(* CODESYS project Kurgan.project
   Company: Plinfa
   Title: Burner
   Author: Serhii Surmylo
   Version: 0.0.0.0

Project tree, tasks and I/O mapping:
  MyController : TM241CEC24T/U, Schneider Electric, order no. TM241CEC24T/U, version 4.0.5.9
    application Application
      task MAST (cyclic, interval 20 ms, priority 15, watchdog 100 ms x 1) calls POU_test
      global variables GVL
      program POU_test [LD]
      Symbols
      function block POU [LD]
    DI : Digital Inputs, Schneider Electric, version 4.0.5.9
        input  A1_IW0 : WORD  // IW0
        input  ibDI_IB1 : BYTE  // IB1
    DQ : Digital Outputs, Schneider Electric, version 4.0.5.9
        output A1_QW0 : WORD  // QW0
        output qbDQ_QB1 : BYTE  // QB1
    Counters : Counters, Schneider Electric, version 4.0.5.9
    Pulse_Generators : Pulse Generators, Schneider Electric, version 4.0.5.9
    Cartridge_1 : Cartridge, Schneider Electric, version 4.0.5.9
    IO_Bus : IO bus - TM3, Schneider Electric, version 4.0.5.9
      A3 : TM2AMI8HT, Schneider Electric, order no. TM2AMI8HT, version 3.1.2.14
          input  A3_IW0 : INT  // IW0
          input  A3_IW1 : INT  // IW1
          input  A3_IW2 : INT  // IW2
          input  A3_IW3 : INT  // IW3
          input  A3_IW4 : INT  // IW4
          input  A3_IW5 : INT  // IW5
          input  A3_IW6 : INT  // IW6
          input  A3_IW7 : INT  // IW7
      A4 : TM2AMI8HT, Schneider Electric, order no. TM2AMI8HT, version 3.1.2.14
          input  A4_IW0 : INT  // IW0
          input  A4_IW1 : INT  // IW1
          input  A4_IW2 : INT  // IW2
          input  A4_IW3 : INT  // IW3
          input  A4_IW4 : INT  // IW4
          input  A4_IW5 : INT  // IW5
          input  A4_IW6 : INT  // IW6
          input  A4_IW7 : INT  // IW7
      A2 : TM3DQ32TK, Schneider Electric, order no. TM3DQ32TK, version 1.0.1.2
          output A2_QD1 : DWORD  // QD0
      A5 : TM2ARI8LT, Schneider Electric, order no. TM2ARI8LT, version 3.1.1.14
          input  A5_IW0 : INT  // IW0
          input  A5_IW1 : INT  // IW1
          input  A5_IW2 : INT  // IW2
          input  A5_IW3 : INT  // IW3
          input  A5_IW4 : INT  // IW4
          input  A5_IW5 : INT  // IW5
          input  A5_IW6 : INT  // IW6
          input  A5_IW7 : INT  // IW7
    COM_Bus : COM bus, Schneider Electric, version 4.0.5.9
    Ethernet_1 : Ethernet Network, Schneider Electric, version 4.0.5.9
        settings: IPAddress = [192, 168, 0, 10]; SubnetMask = [255, 255, 255, 0]; GatewayAddress = [192, 168, 0, 1]; WebServer = TRUE; FTP Server = TRUE; SoMachine Protocol = TRUE; Modbus Server = TRUE; NetManage Protocol = TRUE; SNMP protocol = TRUE; Enable Routing = FALSE; WebVisu protocol = TRUE; DHCP Server Active = TRUE
    Serial_Line_1 : Serial line, Schneider Electric, version 4.0.5.9
    Serial_Line_2 : Serial line, Schneider Electric, version 4.0.5.9
    CAN_1 : CANopen bus, Schneider Electric, version 4.0.5.9
  HMIGTO5310_5315 : HMIGTO5310/5315, Schneider Electric, order no. HMIGTO5310/5315, version 3.5.3.55
    HMI Application
    COM1
      SoMachine_Network_Manager : SoMachine-Network Manager, Schneider Electric, version 4.0.0.2
    COM2
      SoMachine_Network_Manager1 : SoMachine-Network Manager, Schneider Electric, version 4.0.0.2
    Ethernet
      SoMachine_Network_Manager2 : SoMachine-Network Manager, Schneider Electric, version 4.0.0.2
    USB
      SoMachine_Network_Manager3 : SoMachine-Network Manager, Schneider Electric, version 4.0.0.2
  program POU_modbus_SINGLE_WRITE [LD]
  program POU_modbus_READ_VAR [LD]
  program POU_modbus_WRITE_VAR_bit [FBD]
  Vijeo Designer Project Container Data
  Vijeo Designer Project Container
*)

// MyController/Application/GVL
VAR_GLOBAL
END_VAR
VAR_GLOBAL
	KLxx_0_1: BOOL;
	KLxx_ON_OFF: BOOL;
END_VAR

// MyController/Application/POU_test
PROGRAM POU_test
VAR // added by the converter: edge detectors and wires of the graphical bodies
    _rt1, _rt2, _rt3, _rt4 : R_TRIG;
    _ft1, _ft2, _ft3, _ft4 : F_TRIG;
END_VAR

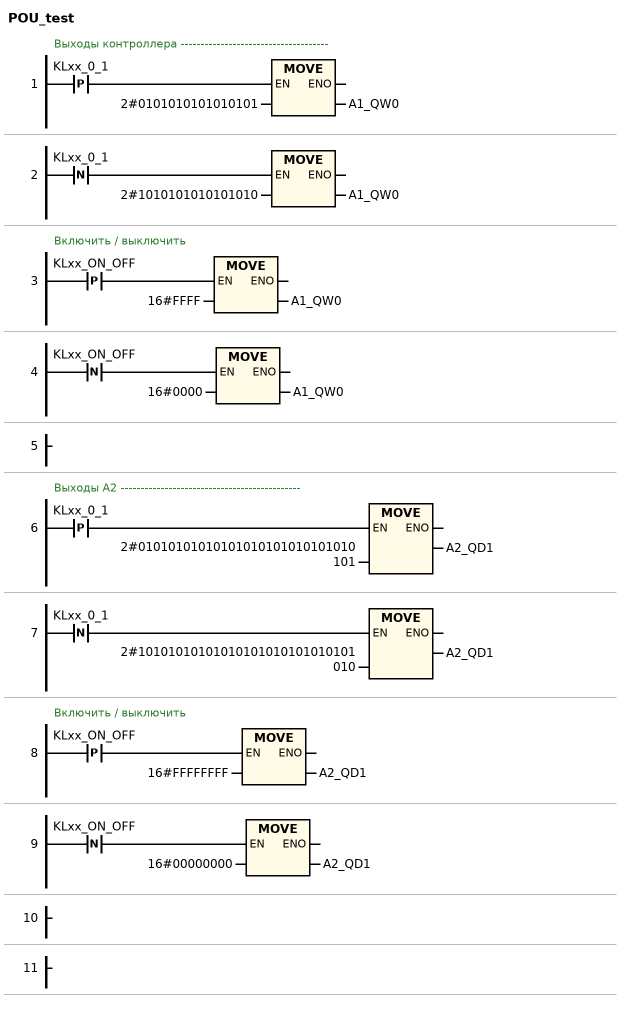
// NETWORK 1
// Выходы контроллера -------------------------------------
//   A1_QW0: DQ : | AT %QW0
_rt1(CLK := KLxx_0_1);
IF _rt1.Q THEN A1_QW0 := 2#0101010101010101; END_IF

// NETWORK 2
//   A1_QW0: DQ : | AT %QW0
_ft1(CLK := KLxx_0_1);
IF _ft1.Q THEN A1_QW0 := 2#1010101010101010; END_IF

// NETWORK 3
// Включить / выключить
//   A1_QW0: DQ : | AT %QW0
_rt2(CLK := KLxx_ON_OFF);
IF _rt2.Q THEN A1_QW0 := 16#FFFF; END_IF

// NETWORK 4
//   A1_QW0: DQ : | AT %QW0
_ft2(CLK := KLxx_ON_OFF);
IF _ft2.Q THEN A1_QW0 := 16#0000; END_IF

// NETWORK 5

// NETWORK 6
// Выходы A2 ---------------------------------------------
//   A2_QD1: A3 : | AT %QD1
_rt3(CLK := KLxx_0_1);
IF _rt3.Q THEN A2_QD1 := 2#01010101010101010101010101010101; END_IF

// NETWORK 7
//   A2_QD1: A3 : | AT %QD1
_ft3(CLK := KLxx_0_1);
IF _ft3.Q THEN A2_QD1 := 2#10101010101010101010101010101010; END_IF

// NETWORK 8
// Включить / выключить
//   A2_QD1: A3 : | AT %QD1
_rt4(CLK := KLxx_ON_OFF);
IF _rt4.Q THEN A2_QD1 := 16#FFFFFFFF; END_IF

// NETWORK 9
//   A2_QD1: A3 : | AT %QD1
_ft4(CLK := KLxx_ON_OFF);
IF _ft4.Q THEN A2_QD1 := 16#00000000; END_IF

// NETWORK 10

// NETWORK 11

END_PROGRAM

// POU_modbus_SINGLE_WRITE
PROGRAM POU_modbus_SINGLE_WRITE
VAR
	temp_var: BOOL;
	res_var: BOOL;
	ADDM_REG0: ADDM;
	SLI_Slave_addr: ADDRESS;
	start: BOOL;
	READ_VAR_REG0: READ_VAR;
	ReceiveBuffer: ARRAY [0..6] OF WORD;
	
	MV1_from_slave8 : WORD;
	MV2_from_slave8 : WORD;
	BLINK_0: BLINK;
	SINGLE_WRITE_REG0: SINGLE_WRITE;
	inc_val: WORD := 705;
	go: BOOL;
END_VAR
VAR // added by the converter: edge detectors and wires of the graphical bodies
    _rt1 : R_TRIG;
    _w1 : BOOL;
END_VAR

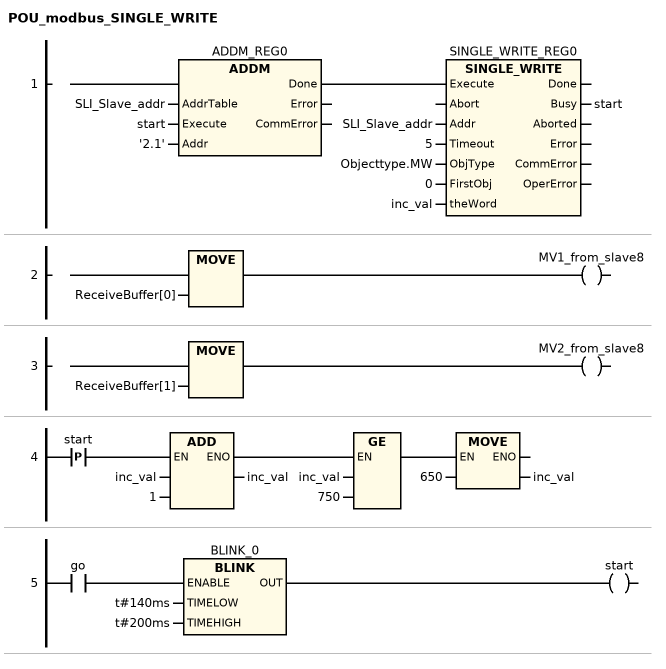
// NETWORK 1
//   Objecttype.MW: Internal Register
ADDM_REG0(AddrTable := SLI_Slave_addr, Execute := start, Addr := '2.1'); // ADDM
SINGLE_WRITE_REG0(
    Execute := ADDM_REG0.Done,
    Addr := SLI_Slave_addr,
    Timeout := 5,
    ObjType := Objecttype.MW,
    FirstObj := 0,
    theWord := inc_val,
    Busy => start); // SINGLE_WRITE

// NETWORK 2
MV1_from_slave8 := ReceiveBuffer[0];

// NETWORK 3
MV2_from_slave8 := ReceiveBuffer[1];

// NETWORK 4
_rt1(CLK := start);
_w1 := _rt1.Q;
IF _w1 THEN inc_val := inc_val + 1; END_IF
IF _w1 AND inc_val >= 750 THEN inc_val := 650; END_IF

// NETWORK 5
BLINK_0(ENABLE := go, TIMELOW := t#140ms, TIMEHIGH := t#200ms); // BLINK
start := BLINK_0.OUT;

END_PROGRAM

// POU_modbus_READ_VAR
PROGRAM POU_modbus_READ_VAR
VAR
	temp_var: BOOL;
	res_var: BOOL;
	ADDM_REG0: ADDM;
	SLI_Slave_addr: ADDRESS;
	start: BOOL;
	READ_VAR_REG0: READ_VAR;
	ReceiveBuffer: ARRAY [0..4] OF WORD;
	BLINK_0: BLINK;
	go: BOOL;
END_VAR

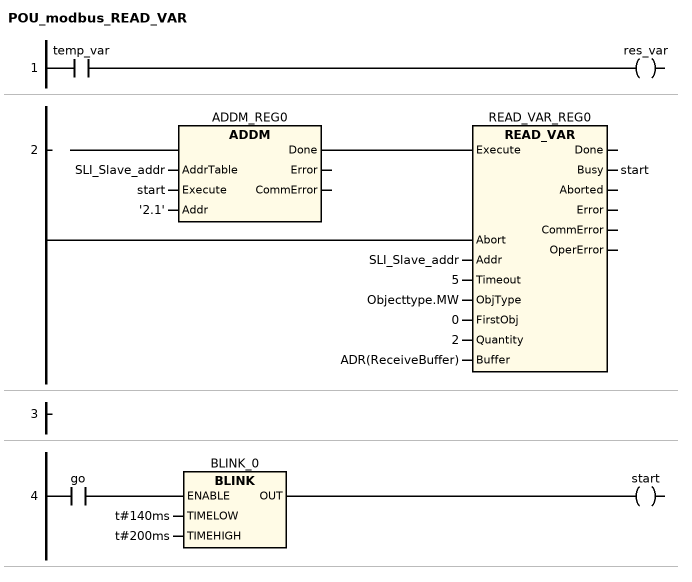
// NETWORK 1
res_var := temp_var;

// NETWORK 2
//   Objecttype.MW: Internal Register
ADDM_REG0(AddrTable := SLI_Slave_addr, Execute := start, Addr := '2.1'); // ADDM
READ_VAR_REG0(
    Execute := ADDM_REG0.Done,
    Abort := TRUE,
    Addr := SLI_Slave_addr,
    Timeout := 5,
    ObjType := Objecttype.MW,
    FirstObj := 0,
    Quantity := 2,
    Buffer := ADR(ReceiveBuffer),
    Busy => start); // READ_VAR

// NETWORK 3

// NETWORK 4
BLINK_0(ENABLE := go, TIMELOW := t#140ms, TIMEHIGH := t#200ms); // BLINK
start := BLINK_0.OUT;

END_PROGRAM

// POU_modbus_WRITE_VAR_bit
PROGRAM POU_modbus_WRITE_VAR_bit
VAR
	ADDM_REG0: ADDM;
	SLI_Slave_addr: ADDRESS;
	start: BOOL;
	SendBuffer: WORD := 1;
	SendBuffer2: ARRAY [0..3] OF WORD;
	BLINK_0: BLINK;
	WRITE_VAR_BIT: WRITE_VAR;
	go: BOOL := TRUE;
END_VAR
VAR // added by the converter: edge detectors and wires of the graphical bodies
    _rt1 : R_TRIG;
    _w1 : BOOL;
END_VAR

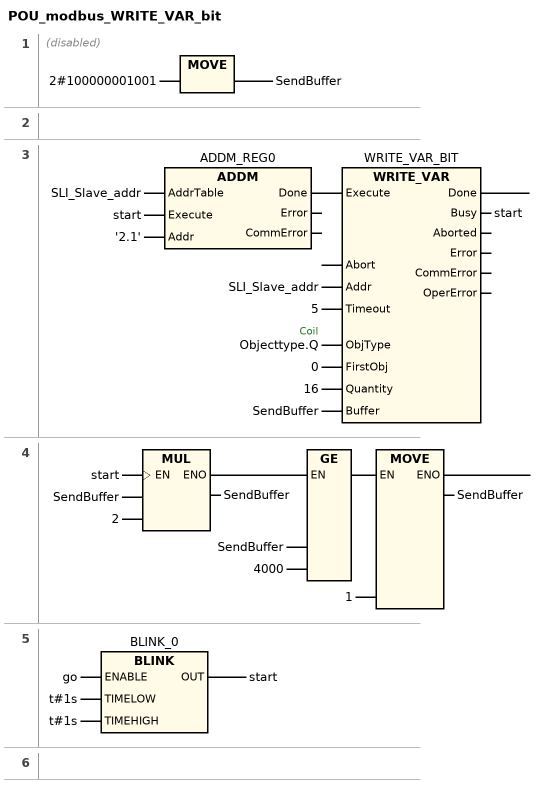
// NETWORK 1 (disabled)
// SendBuffer := 2#100000001001;

// NETWORK 2

// NETWORK 3
//   Objecttype.Q: Coil
ADDM_REG0(AddrTable := SLI_Slave_addr, Execute := start, Addr := '2.1'); // ADDM
WRITE_VAR_BIT(
    Execute := ADDM_REG0.Done,
    Addr := SLI_Slave_addr,
    Timeout := 5,
    ObjType := Objecttype.Q,
    FirstObj := 0,
    Quantity := 16,
    Buffer := SendBuffer,
    Busy => start); // WRITE_VAR

// NETWORK 4
_rt1(CLK := start);
_w1 := _rt1.Q;
IF _w1 THEN SendBuffer := SendBuffer * 2; END_IF
IF _w1 AND SendBuffer >= 4000 THEN SendBuffer := 1; END_IF

// NETWORK 5
BLINK_0(ENABLE := go, TIMELOW := t#1s, TIMEHIGH := t#1s); // BLINK
start := BLINK_0.OUT;

// NETWORK 6

END_PROGRAM

// MyController/Application/POU
FUNCTION_BLOCK POU
VAR_INPUT
	q1: BOOL;
END_VAR
VAR_OUTPUT
	out1: BOOL;
END_VAR
VAR
END_VAR

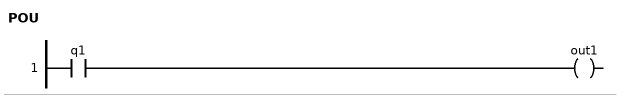
// NETWORK 1
out1 := q1;

END_FUNCTION_BLOCK
